KUKA KRL program: chk_w6_grp2_clo.src

&ACCESS RVO1
&COMMENT Accelo Z2.1_Z2.2
DEF chk_w6_grp2_clo( )

; Check gripper ACCELO CLOSE Z2.1 Z2.2

$TIMER[10] = 0
$TIMER_STOP[10] = FALSE

WAIT FOR (NOT $IN[37] AND NOT $IN[39] AND NOT $IN[41])
WAIT FOR ($IN[38] AND $IN[40] AND $IN[42])

$TIMER_STOP[10] = TRUE
$TIMER[10] = 0

;//---- Start User-------
;//---- End User---------
END
